INTERFACE I_Callable

METHOD Call
VAR_INPUT
	iArg		: I_Arg;
END_VAR
END_METHOD

END_INTERFACE

(* stored: Version 1.1.0.1
   Itf I_Callable: Id {12666b7d-e29e-43ef-8ad6-3108c77eb213}
   Method Call: Id {8832ca44-0762-4c0a-bb8a-499db047863a} *)
